	// Config Values 
	mcHomingMode 		: MC_HomingMode ; 
	fHomePosition		: LREAL := 0 ; // set position at homing
	fSafeVeloLimit		: LREAL	:= 360 ; // safe velocity limit [deg/sec]
	nEncTurnoverVal 	: LREAL ; // encoder turnover value 
	tDisabledelay		: TIME 	; // Axis idle time before axis is disabled 
END_VAR
VAR 
	bActVeloReadValid 	: BOOL ; // velocity parameter read is valid 
	bActAccReadValid 	: BOOL ; // Acceleration parameter read is valid 
	bActDecReadValid 	: BOOL ; // Deceleration parameter read is valid 
	bActParamValid 		: BOOL ; // Parameter read is valid 
END_VAR
// ===== Message data set =====
	stFault.LocationName  	:= sName 	;
	stFault.LocationNumber 	:= sNumber 	;
	stFault.ComponentType		:= E_ComponentTypes.Axis ;
	
// ===== Read system configuration =====
	McReadSysVelo	(	Axis 			:= AxisRef,
						Enable 			:= Cmd_EnDriveParRead ,
						ParameterNumber := MaxVelocitySystem ,
						ReadMode		:= 1,
						Valid			=> bActVeloReadValid ,						
						Busy			=> ,
						Error			=> ,
						ErrorID			=> ,
						Value			=> fMaxVelo );
	McReadSysAcc	(	Axis 			:= AxisRef,
						Enable 			:= Cmd_EnDriveParRead ,
						ParameterNumber := MaxAccelerationSystem ,
						ReadMode		:= 1,
						Valid			=> bActAccReadValid ,						
						Busy			=> ,
						Error			=> ,
						ErrorID			=> ,
						Value			=> fMaxAcc );
	McReadSysDec	(	Axis 			:= AxisRef,
						Enable 			:= Cmd_EnDriveParRead ,
						ParameterNumber := MaxDecelerationSystem ,
						ReadMode		:= 1,
						Valid			=> bActDecReadValid ,						
						Busy			=> ,
						Error			=> ,
						ErrorID			=> ,
						Value			=> fMaxDec );

	IF 	fMaxVelo > 0 
	AND fMaxAcc >0
	AND fMaxDec >0 THEN 
		bActParamValid	:= TRUE ; 
		fCmdAcc 		:= fMaxAcc * 0.9;
		fCmdDecc		:= fMaxDec * 0.9;
	END_IF

	IF NOT Cmd_EnDriveParRead AND NOT bActParamValid THEN  
		Cmd_EnDriveParRead := TRUE;
	ELSIF Cmd_EnDriveParRead THEN
		Cmd_EnDriveParRead := FALSE;
	END_IF

// ===== Configure Axis =====
	// ***** Config Bits *****
		THIS^.bIcfCmdVelocityRpm	:= bIcfCmdVelocityRpm	; // Enable speed inputs in Rpm
		THIS^.bIcfEnableForward 	:= bIcfEnableForward 	; // Enable forward motion
		THIS^.bIcfEnablereverse		:= bIcfEnablereverse	; // Enable reverse motion
		THIS^.bIcfAlwaysEnable		:= bIcfAlwaysEnable		; // Always enable motor and brake if safety is ok
	// ***** config homing Mode ***** 
 		THIS^.mcHomingMode 			:= mcHomingMode ; // set homing mode
		THIS^.fHomePosition			:= fHomePosition;
	// ***** Velocity settings *****
		THIS^.fSafeVeloLimit 		:= fSafeVeloLimit ; // set maximum safe velocity	
	// ***** Encoder values *****
		THIS^.fEncoderTurnoverValue := nEncTurnoverVal	; // turnover value for encoder = 25.6 mm per rev * 4096 revolutions 
	// ***** Time delay enable off *****
		THIS^.tDisableDelay 	:= tDisabledelay ;		

// ===== reset axis state indicators ======
	bError 	:= FALSE;

// ====== Set init to done =======
IF bActParamValid THEN 
	bInitDone	:= TRUE ; 
END_IF
END_METHOD

METHOD PRIVATE ExecGearDynamic : BOOL
VAR_INPUT
END_VAR
// ===== invert gear ratio if reverse slave is active =====
	IF bReverseSlave THEN 
		fbMcGearInDyn.GearRatio := fCmdGearRatio * -1 ;
	ELSE 
		fbMcGearInDyn.GearRatio := fCmdGearRatio ;
	END_IF

// ===== Execute gear in function =====
	fbMcGearInDyn ( 	Master 			:= refMasterAxis,
						Slave			:= AxisRef,
						Enable 			:= bExec_GearSlaveDyn,
						Acceleration	:= fCmdAcc	); 
						
// ===== reset command =====
	bGearedAsSlave		:= fbMcGearInDyn.InGear ; 

// Gearing fault handling 
	IF fbMcGearInDyn.Error THEN 
		bError					:= TRUE							;
		stFault.Active 			:= TRUE 						;
		stFault.MessageNumber	:= E_MessageNumbers.FF_AxisFault;
		stFault.Discription		:= CONCAT('Gear dynamic Fault ', UDINT_TO_STRING(fbMcGearInDyn.ErrorID));				;
		stFault.FaultType		:= E_FaultTypes.FF				;
		refFbFault.CmdAddFault( stFault );
	END_IF
END_METHOD

METHOD PRIVATE ExecGearIn : BOOL
VAR_INPUT
END_VAR
// ===== invert gear ratio if reverse slave is active =====
	IF bReverseSlave THEN 
		fbMcGearInSlave.RatioNumerator := fCmdGearRatio * -1 ;
	ELSE 
		fbMcGearInSlave.RatioNumerator := fCmdGearRatio ;
	END_IF

// ===== Execute gear in function =====
	fbMcGearInSlave ( 	Master 			:= refMasterAxis,
						Slave			:= AxisRef,
						Execute 		:= bExec_GearAsSlave,
						RatioDenominator:= 1	); 
						
// ===== reset command =====
	bExec_GearAsSlave 	:= FALSE  ;
	bGearedAsSlave		S= fbMcGearInSlave.InGear ; 

// Gearing fault handling 
	IF fbMcGearInSlave.Error THEN 
		bError					:= TRUE							;
		stFault.Active 			:= TRUE 						;
		stFault.MessageNumber	:= E_MessageNumbers.FF_AxisFault;
		stFault.Discription		:= CONCAT('Gear as slave Fault ', UDINT_TO_STRING(fbMcGearInSlave.ErrorID));				;
		stFault.FaultType		:= E_FaultTypes.FF				;
		refFbFault.CmdAddFault( stFault );
	END_IF
END_METHOD

METHOD PRIVATE ExecGearOut : BOOL
VAR_INPUT
END_VAR
// ===== execute gear out function ======
	fbMcGearOutSlave (	Slave 	:= AxisRef,
						Execute := bExec_GearOutSlave );

// ===== reset command =====
	bExec_GearOutSlave	:= false ;
	bGearedAsSlave		R= fbMcGearOutSlave.Done 	; 

// Gearing fault handling 
	IF fbMcGearOutSlave.Error THEN 
		bError					:= TRUE							;
		stFault.Active 			:= TRUE 						;
		stFault.MessageNumber	:= E_MessageNumbers.FF_AxisFault;
		stFault.Discription		:= CONCAT('Gear out Fault ', UDINT_TO_STRING(fbMcGearOutSlave.ErrorID));				;
		stFault.FaultType		:= E_FaultTypes.FF				;
		refFbFault.CmdAddFault( stFault );
	END_IF
END_METHOD

METHOD PRIVATE ExecHalt : BOOL
VAR_INPUT
END_VAR
// ==== Execute halt function ===== 
fbMcHalt (	Axis 		:= AxisRef,
			Execute 	:= bExec_Halt );

// ===== reset command =====
	bExec_Halt := FALSE ;
	
// Halt fault handling 
	IF fbMcHalt.Error THEN 
		bError					:= TRUE							;
		stFault.Active 			:= TRUE 						;
		stFault.MessageNumber	:= E_MessageNumbers.FF_AxisFault;
		stFault.Discription		:= CONCAT('Halt Fault ', UDINT_TO_STRING(fbMcHalt.ErrorID));				;
		stFault.FaultType		:= E_FaultTypes.FF				;
		refFbFault.CmdAddFault( stFault );
	END_IF
END_METHOD

METHOD PRIVATE ExecHome : BOOL
VAR_INPUT
END_VAR
// ==== execute homing function =====
	fbMcHome(	Axis			:= AxisRef,
				Execute			:= bExec_Home,
				HomingMode		:= mcHomingMode,
				bCalibrationCam	:= IAxisHome ); 
			
// Reset exec command 
	bExec_Home 	:= FALSE ;
	bHomed		S= fbMcHome.Done ;	
				
// fault handling 
	IF fbMcHome.Error THEN 
		bError					:= TRUE							;
		stFault.Active 			:= TRUE 						;
		stFault.MessageNumber	:= E_MessageNumbers.FF_AxisFault;
		stFault.Discription		:= CONCAT('Homing Fault ', UDINT_TO_STRING(fbMcHome.ErrorID));				;
		stFault.FaultType		:= E_FaultTypes.FF				;
		refFbFault.CmdAddFault( stFault );
	END_IF
END_METHOD

METHOD PRIVATE ExecJog : BOOL
VAR_INPUT
END_VAR
// ===== Execute Jog function =====
	// velocity limiting
		IF bCmdSafeSpeed THEN 
			fbMcJog.Velocity := MIN(fSafeVeloLimit, fbMcJog.Velocity); 
		ELSIF bCmdLimitVelocity THEN 
			fbMcJog.Velocity := MIN(fCmdVelocityLimit, fbMcJog.Velocity); 
		END_IF
	// function call
	fbMcJog (	Axis 		:= AxisRef,
				JogForward	:= bExec_JogPositive,
				JogBackwards:= bExec_JogNegative,
				Acceleration:= fCmdAcc,
				Deceleration:= fCmdDecc );

// ===== reset command =====
	bExec_JogPositive 	:= FALSE  ;
	bExec_JogNegative	:= FALSE  ;
	
// Jog fault handling 
	IF fbMcJog.Error THEN 
		bError					:= TRUE							;
		stFault.Active 			:= TRUE 						;
		stFault.MessageNumber	:= E_MessageNumbers.FF_AxisFault;
		stFault.Discription		:= CONCAT('Jog Fault ', UDINT_TO_STRING(fbMcJog.ErrorID));				;
		stFault.FaultType		:= E_FaultTypes.FF				;
		refFbFault.CmdAddFault( stFault );
	END_IF
END_METHOD

METHOD PRIVATE ExecMoveAbsolute : BOOL
VAR_INPUT
END_VAR
// ==== execute move absolute function =====
FOR i := 0 TO 1 DO 
	// velocity limiting
		IF bCmdSafeSpeed THEN 
			fbMcMoveAbsolute[i].Velocity := MIN(fSafeVeloLimit, fbMcMoveAbsolute[i].Velocity); 
		ELSIF bCmdLimitVelocity THEN 
			fbMcMoveAbsolute[i].Velocity := MIN(fCmdVelocityLimit, fbMcMoveAbsolute[i].Velocity); 
		END_IF
	// function call
	fbMcMoveAbsolute[i](	Axis 		:= AxisRef,
							Execute 	:= arExec_MoveAbs[i],
							Acceleration:= fCmdAcc,
							Deceleration:= fCmdDecc );  
	// reset Exec command 
	arExec_MoveAbs[i] := FALSE ; 

	// If function is done then reset command values
	IF fbMcMoveAbsolute[i].Done THEN 
		fbMcMoveAbsolute[i].Velocity	:= 0 ;
		fbMcMoveAbsolute[i].Position	:= 0 ; 
	END_IF
	
	// fault handling 
	IF fbMcMoveAbsolute[i].Error THEN 
		bError					:= TRUE							;
		stFault.Active 			:= TRUE 						;
		stFault.MessageNumber	:= E_MessageNumbers.FF_AxisFault;
		stFault.Discription		:= CONCAT('Move absolute Fault ', UDINT_TO_STRING(fbMcMoveAbsolute[i].ErrorID));				;
		stFault.FaultType		:= E_FaultTypes.FF				;
		refFbFault.CmdAddFault( stFault );
	END_IF
END_FOR
END_METHOD

METHOD PRIVATE ExecMoveModulo : BOOL
VAR_INPUT
END_VAR
// ===== Execute move modulo function =====
FOR i := 0 TO 1 DO 
	// velocity limiting
		IF bCmdSafeSpeed THEN 
			fbMcMoveModulo[i].Velocity := MIN(fSafeVeloLimit, fbMcMoveModulo[i].Velocity); 
		ELSIF bCmdLimitVelocity THEN 
			fbMcMoveModulo[i].Velocity := MIN(fCmdVelocityLimit, fbMcMoveModulo[i].Velocity); 
		END_IF
	// function call
	fbMcMoveModulo[i](	Axis 		:= AxisRef,
						Execute 	:= arExec_MoveModulo[i],
						Acceleration:= fCmdAcc,
						Deceleration:= fCmdDecc);  
	// reset Exec command 
	arExec_MoveModulo[i] := FALSE ; 
	
	// If function is done then reset command values
	IF fbMcMoveModulo[i].Done THEN 
		fbMcMoveModulo[i].Velocity	:= 0 ;
		fbMcMoveModulo[i].Position	:= 0 ; 
	END_IF
	
	// fault handling 
	IF fbMcMoveModulo[i].Error THEN 
		bError					:= TRUE							;
		stFault.Active 			:= TRUE 						;
		stFault.MessageNumber	:= E_MessageNumbers.FF_AxisFault;
		stFault.Discription		:= CONCAT('Move module Fault ', UDINT_TO_STRING(fbMcMoveModulo[i].ErrorID));				;
		stFault.FaultType		:= E_FaultTypes.FF			;
		refFbFault.CmdAddFault( stFault );
	END_IF
END_FOR
END_METHOD

METHOD PRIVATE ExecMoveRelative : BOOL
VAR_INPUT
END_VAR
// ===== Execute move relative function ======
FOR i := 0 TO 1 DO 
	// velocity limiting
		IF bCmdSafeSpeed THEN 
			fbMCMoveRelative[i].Velocity := MIN(fSafeVeloLimit, fbMCMoveRelative[i].Velocity); 
		ELSIF bCmdLimitVelocity THEN 
			fbMCMoveRelative[i].Velocity := MIN(fCmdVelocityLimit, fbMCMoveRelative[i].Velocity); 
		END_IF
	// function call
	fbMCMoveRelative[i](	Axis 		:= AxisRef,
							Execute		:= arExec_MoveRelative[i],
							Acceleration:= fCmdAcc,
							Deceleration:= fCmdDecc );
	// reset Exec command 
	arExec_MoveRelative[i] := FALSE ; 

	// If function is done then reset command values
	IF fbMCMoveRelative[i].Done THEN 
		fbMCMoveRelative[i].Velocity	:= 0 ;
		fbMCMoveRelative[i].Distance	:= 0 ; 
	END_IF
	
	// fault handling 
	IF fbMCMoveRelative[i].Error THEN 
		bError					:= TRUE							;
		stFault.Active 			:= TRUE 						;
		stFault.MessageNumber	:= E_MessageNumbers.FF_AxisFault;
		stFault.Discription		:= CONCAT('Move relative Fault ', UDINT_TO_STRING(fbMCMoveRelative[i].ErrorID));				;
		stFault.FaultType		:= E_FaultTypes.FF			;
		refFbFault.CmdAddFault( stFault );
	END_IF
END_FOR
END_METHOD

METHOD PRIVATE ExecMoveVelocity : BOOL
VAR_INPUT
END_VAR
// ===== Execute move velocity function =====
// velocity limiting
IF bCmdSafeSpeed THEN 
	fbMcMoveVelocity.Velocity := MIN(fSafeVeloLimit, fbMcMoveVelocity.Velocity); 
ELSIF bCmdLimitVelocity THEN 
	fbMcMoveVelocity.Velocity := MIN(fCmdVelocityLimit, fbMcMoveVelocity.Velocity); 
END_IF
// function call
fbMcMoveVelocity (	Axis 		:= AxisRef,
					Execute		:= bExec_MoveVelocity,
					Acceleration:= fCmdAcc,
					Deceleration:= fCmdDecc );

// ===== reset command =====
bExec_MoveVelocity := FALSE ;
	
// Halt fault handling 
IF fbMcHalt.Error THEN 
	bError					:= TRUE							;
	stFault.Active 			:= TRUE 						;
	stFault.MessageNumber	:= E_MessageNumbers.FF_AxisFault;
	stFault.Discription		:= CONCAT('Move velocity Fault ', UDINT_TO_STRING(fbMcMoveVelocity.ErrorID));				;
	stFault.FaultType		:= E_FaultTypes.FF				;
	refFbFault.CmdAddFault( stFault );
END_IF
END_METHOD

METHOD PRIVATE ExecEnable : BOOL
VAR_INPUT
END_VAR
// ===== Set axis enable ======
IF NOT bEnable AND NOT AxisRef.Status.MotionCommandsLocked THEN
	bCmdSafeStop	S= TRUE ;
ELSE 
	bCmdEnableAxis	:= bEnable ;
END_IF

// ===== Check if axis is bussy with a command =====
	bInternalEnable S= AxisRef.Status.HasJob;
	bInternalEnable	S= bIcfAlwaysEnable ; // always enable axis if configured
	bInternalEnable	S= AxisRef.Status.Coupled ;
	
// ===== Axis disable timer after last command =====
	TofIntAxisEnable (	IN:= bInternalEnable, PT := tDisableDelay);

// ===== Enable drive =====
	fbMcPower(	Axis			:= AxisRef , 
				Enable			:= bCmdEnableAxis AND TofIntAxisEnable.Q, 
				Enable_Positive	:= bIcfEnableForward, 
				Enable_Negative	:= bIcfEnablereverse, 
				Override		:= 100 );  
				
// ===== Reset internal enable signal =====
	bInternalEnable := FALSE ; 	

IF fbMcPower.Error THEN 
	bError					:= TRUE							;
	stFault.Active 			:= TRUE 						;
	stFault.MessageNumber	:= E_MessageNumbers.FF_AxisFault;
	stFault.Discription		:= CONCAT('Enable Fault ', UDINT_TO_STRING(fbMcPower.ErrorID));				;
	stFault.FaultType		:= E_FaultTypes.FF				;
	refFbFault.CmdAddFault( stFault );
END_IF
END_METHOD

METHOD PRIVATE ExecReadStatus : BOOL
VAR_INPUT
END_VAR
// Read axis status from drive
fbMcReadAxisStatus (	Enable 	:= TRUE ,
						Axis 	:= AxisRef );
						
// convert velocity to RPM for output if aplicable
IF bIcfCmdVelocityRpm THEN 
	fVelocity := AxisRef.NcToPlc.ActVelo / 6 ;
ELSE 
	fVelocity := AxisRef.NcToPlc.ActVelo ;
END_IF
						
// set status bits 
bIdle := NOT AxisRef.Status.HasJob ;

// read fault handling 
IF fbMcReadAxisStatus.Error THEN 
	bError					:= TRUE							;
	stFault.Active 			:= TRUE 						;
	stFault.MessageNumber	:= E_MessageNumbers.FF_AxisFault;
	stFault.Discription		:= CONCAT('Status read fault ', UDINT_TO_STRING(fbMcPower.ErrorID));				;
	stFault.FaultType		:= E_FaultTypes.FF				;
	refFbFault.CmdAddFault( stFault );
END_IF
END_METHOD

METHOD PRIVATE ExecReset : BOOL
VAR_INPUT
END_VAR
IF  AxisRef.Status.Moving THEN // If the axis is still moving execute safe stop first
	CmdSafeStop();
	RETURN;
END_IF

// ===== Reset axis, drive and axis functions =====
	fbSoeReset ( 	Execute := bExec_Reset AND NOT fbMcReset.Busy AND NOT bIcfSimulationMode, // No physical drive reset necesarry when not connected 
					Timeout := T#10S		,
					Axis	:= AxisRef		);
	
	fbMcReset	( 	Execute	:= bexec_reset AND NOT fbSoeReset.Busy,
					Axis	:= AxisRef ); 
					
// ===== reset command =====
	bExec_Reset := FALSE ;
	
// ===== reset internal fault bits and stop bits =====
	bError 			:= FALSE ; 
	
// ===== reset safe commands ======
	bCmdSafeStop	:= FALSE ; 
	bCmdSafeSpeed 	:= FALSE ;
	
// Reset fault handling 
	IF fbSoeReset.Error OR fbMcReset.Error THEN 
		bError					:= TRUE							;
		stFault.Active 			:= TRUE 						;
		stFault.MessageNumber	:= E_MessageNumbers.FF_AxisFault;
		stFault.Discription		:= CONCAT('Reset Fault ', UDINT_TO_STRING(fbMcReset.ErrorID))			;
		stFault.FaultType		:= E_FaultTypes.FF				;
		refFbFault.CmdAddFault( stFault );
	END_IF
END_METHOD

METHOD PRIVATE ExecSafeFunctions : BOOL
VAR_INPUT
END_VAR
// ==== Safe operation functions (overrule all other motion functions) =====
	fbMcStop( 	Axis 			:= AxisRef		,
				Execute 		:= bCmdSafeStop	,
				Deceleration	:= fMaxDec		);
	
	// Reset axis command			
	bCmdSafeStop 	R= fbMcStop.Done OR AxisRef.Status.HasBeenStopped ;
	bStopped		:= AxisRef.Status.HasBeenStopped ;
	
// Safestop fault handling 
	IF fbMcStop.Error THEN 
		bError					:= TRUE							;
		stFault.Active 			:= TRUE 						;
		stFault.MessageNumber	:= E_MessageNumbers.FF_AxisFault;
		stFault.Discription		:= CONCAT('Safe stop axis fault ', UDINT_TO_STRING(fbMcStop.ErrorID));				;
		stFault.FaultType		:= E_FaultTypes.FF				;
		refFbFault.CmdAddFault( stFault );
	END_IF
	
// ===== Safe speed monitoring =====
	IF bCmdSafeSpeed THEN 
		IF AxisRef.NcToPlc.ActVelo > fSafeVeloLimit THEN 
			bExec_Halt := TRUE ; 
			ExecHalt(); 
		ELSE 
			bCmdSafeSpeed := FALSE ; 
		END_IF
	END_IF

// ===== Dev is safe feedback =====
bDevIsSafe := AxisRef.Status.HasBeenStopped AND NOT bCmdEnableAxis ;
END_METHOD

METHOD PRIVATE METH_ExecuteMotionFunctions : BOOL
VAR_INPUT
END_VAR
// ===== Check if safe to move =====
	IF bCmdSafeStop THEN 
		RETURN ;
	END_IF

// ===== Homing functions =====
	ExecHome		(); 

// ===== Motion standstil commands =====
	ExecHalt		();

// ===== Motion move functions
	ExecJog			(); 
	ExecMoveAbsolute();
	ExecMoveRelative();
	ExecMoveModulo	();
	ExecMoveVelocity();
	
// ===== Execute gearing functions =====
	ExecGearIn		();
	ExecGearDynamic	();
	ExecGearOut		();
	
// ====== reset velocity lmiting =====
	bVelocityLimited	:= bCmdLimitVelocity ;	
	bCmdLimitVelocity 	:= FALSE ;
END_METHOD

METHOD PRIVATE METH_ExecuteOrganizationFunctions : BOOL
VAR_INPUT
END_VAR
// ==== execute organizational functions =====
	ExecReadStatus	(); 
	ExecEnable		();
	ExecReset		();
END_METHOD

END_FUNCTION_BLOCK

// Buttons/Functions/FB_DevHMIButton
FUNCTION_BLOCK PUBLIC FB_DevHMIButton EXTENDS FB_DevBase // Button function for HMI 
VAR_INPUT
	Istatus			: BOOL	:= FALSE;// Digital sensor, Direct input status
	tDelay			: TIME 	:= T#5S	;// Time before delayed signal becomes active 
	bCmdSimulate	: BOOL 	:= FALSE;// Simulate sensor Input 
	bSimState		: BOOL 	:= FALSE;// Simulated sensor state
END_VAR
VAR_OUTPUT
	bFcoInputActive		: BOOL 			;// Digital sensor, Button active state
	bFcoDelay			: BOOL			;// Button, Delayed input status (3 seconds) 
	bFeStatus			: BOOL			;// Button, Falling edge of input signal	
	bReStatus			: BOOL			;// Button, Rising edge of input signal
	TetInputActive		: TIME			;// Button, Time elapsed while button is active
	bInvisible			: BOOL 			;// Button, Button is made invisible
	bDeactivate			: BOOL 			;// Button, Deactivate button 
END_VAR
VAR
	FB_delIStatus: TON; // Timer function for delayed input status 
	FB_feIStatus: F_TRIG; // generate falling edge pulse edge from Istatus
	FB_reIStatus: R_TRIG; // generate falling edge pulse edge from Istatus
END_VAR

// ***** Direct input when enabled *****
IF bEnable THEN 
	IF bCmdSimulate  THEN 
		bFcoInputActive := bSimState ; 
	ELSE
		bFcoInputActive := Istatus ;
	END_IF
ELSE 
	bFcoInputActive := FALSE ;
END_IF

// ===== check if function is enabled =====
	IF NOT bEnable THEN 
		bInvisible 	:= TRUE ;
		bDeactivate	:= TRUE ;
		bFcoDelay	:= FALSE;
		RETURN;
	ELSE  
		bInvisible 	:= FALSE ;
		bDeactivate	:= FALSE ;
	END_IF

// ====== process functions if enabled ======
	// ***** Set Delayed inputs and time elapsed ****
		FB_delIStatus(	IN:= bFcoInputActive,
						PT:= tDelay , 
						Q=> bFcoDelay , 
						ET=> TetInputActive 
					  ); // Generate delayed input status from push button input status
	// ***** Edge triggers *****
		FB_feIStatus(CLK:= Istatus , Q=> bFeStatus ); // generate falling edge pulse on pushbutton input
		FB_reIStatus (Clk := Istatus , Q => bReStatus); // Generate rising edge from push button input signal

END_FUNCTION_BLOCK

// Buttons/Functions/FB_DevPushButton
FUNCTION_BLOCK PUBLIC FB_DevPushButton EXTENDS Fb_DevDigitalInputFunctions
VAR_INPUT
END_VAR
VAR_OUTPUT
END_VAR
VAR
END_VAR

SUPER^();

END_FUNCTION_BLOCK

// Buttons/Functions/FB_DevPushbuttonLight
FUNCTION_BLOCK PUBLIC FB_DevPushbuttonLight EXTENDS FB_DevPushButton
VAR_INPUT
	sCmdLightState	: E_LightState ; // feedback lights status 
END_VAR
VAR_OUTPUT
END_VAR
VAR
	fbLight : Fb_DevLight ; // light control 
END_VAR

SUPER^();

// Light commands
	CASE sCmdLightState OF
		Light_Off:
			fbLight.eCmdLight := E_LightState.Light_Off;
		Light_BlinkSlow:
			fbLight.eCmdLight := E_LightState.Light_BlinkSlow ;
		Light_BlinkFast:
			fbLight.eCmdLight := E_LightState.Light_BlinkFast ;
		Light_On:
			fbLight.eCmdLight := E_LightState.Light_On ;
	END_CASE
	
fbLight(bEnable := TRUE);

END_FUNCTION_BLOCK

// Lights/Functions/Fb_DevLight
FUNCTION_BLOCK PUBLIC Fb_DevLight
VAR_INPUT
	bEnable			: BOOL	:= TRUE ;// Enable light
	eCmdLight		: E_LightState := E_LightState.Light_Off ; // commanded light state [Light_off, _On, _BlinkFast, _BlinkSlow]
END_VAR
VAR_OUTPUT
END_VAR
VAR
	qLight AT %Q* : BOOL := FALSE ; // light output
END_VAR

// ===== check if light is enabled ======
	IF NOT bEnable THEN 
		qLight := FALSE ;
		RETURN; 
	END_IF
	
// ===== set light output ======
	Mod_SetOutput();

METHOD PRIVATE Mod_SetOutput : BOOL
VAR_INPUT
END_VAR
// ===== set light output state =====
	CASE eCmdLight OF
		Light_BlinkSlow:
			qLight := Sys_Variables.BlinkSlow ;
		Light_BlinkFast:
			qLight	:= Sys_Variables.BlinkFast ;
		Light_On:
			qLight := TRUE ;
		ELSE
			qLight := FALSE ;
	END_CASE
END_METHOD

END_FUNCTION_BLOCK

// Encoders/FunctionBlocks/FB_EncoderBase
FUNCTION_BLOCK PUBLIC FB_EncoderBase
VAR_INPUT
	nCfgUnitsPerPulse	: LREAL := 1	; // Scale factor for output [units/pulse]
	nCfgOffset			: LREAL := 0	; // Offset for output
	
	bIcfInverted		: BOOL	:= FALSE; // Invert output position = standard false  
END_VAR
VAR_OUTPUT
	nOutPosition		: LREAL	:= 0	; // Scaled position output
	nOutRaw				: UDINT := 0	; // Raw output value	 
	nVelocity			: LREAL	:= 0 	; // Velocity [units/sec]
END_VAR
VAR
END_VAR

METHOD PUBLIC FastTask : BOOL
VAR_INPUT
END_VAR
END_METHOD

END_FUNCTION_BLOCK

// Encoders/FunctionBlocks/FB_EncoderInput
FUNCTION_BLOCK FB_EncoderInput EXTENDS FB_EncoderBase
VAR_INPUT
END_VAR
VAR_OUTPUT
END_VAR
VAR
	iEncoderSignal AT%I*: UDINT ;
	
	nScaledValue		: LREAL ; // Only scaled value for internal use
	nValueWithOffset	: LREAL ; // scaled value with added offset
END_VAR

// ====== Scale Output value ======
	nScaledValue := UDINT_TO_LREAL(iEncoderSignal) * nCfgUnitsPerPulse ;

// ====== Invert ======
	IF bIcfInverted THEN 
		nScaledValue := nScaledValue * -1;
	END_IF
	
// ====== Add offset ======= 
	nValueWithOffset := nScaledValue + nCfgOffset ;

// ====== Set Outputs =======
	nOutPosition 	:= nValueWithOffset ;
	nOutRaw			:= iEncoderSignal	;

METHOD PUBLIC FastTask : BOOL
VAR_INPUT
END_VAR
END_METHOD

END_FUNCTION_BLOCK

// GroupHandlers/ManualControlHandler/FB_DevManualHandler
FUNCTION_BLOCK FB_DevManualHandler
VAR_INPUT
END_VAR
VAR_OUTPUT
END_VAR
VAR
END_VAR

END_FUNCTION_BLOCK

// Heaters/FB_DevPWMGenerator
FUNCTION_BLOCK PUBLIC FB_DevPWMGenerator EXTENDS FB_DevBase
VAR_INPUT
	nPeriodLength		: DINT	:= 2000 	; // desired PWM cycle time length [ms] 
	nDutyCycle 	: DINT	:= 0 		; // percentage of power 
END_VAR
VAR_OUTPUT
END_VAR
VAR
	qbOutput	AT %Q* 	: BOOL 	; // physical output
	bCycleOutput		: BOOL 	; // Cycle output
	tonTimerOn  		: TON 	; // Timer for cycle on
	tofTimerOff			: TOF 	; // timer for cycle off 
	// output commands
	bCmdPWMCycle		: BOOL 	; // run PWM cycle 
	bCmdOn				: BOOL 	; // turn output on permanantly
	
END_VAR

// check for enable
IF NOT bEnable THEN 
	qbOutput := FALSE ;
	RETURN; 
ELSE 
	SUPER^(); 
END_IF

// calculate cycle times 
CalcCycle();
// set outputs
ExecSetOutput();

METHOD PRIVATE CalcCycle : BOOL
VAR_INPUT
END_VAR
// check if dutycycle is within limits
nDutyCycle := LIMIT(1,nDutyCycle,100);

// Calculate time on from cycle time
tonTimerOn.PT 	:= DINT_TO_TIME(( nPeriodLength / 100) * nDutyCycle);
tofTimerOff.PT	:= DINT_TO_TIME(( nPeriodLength / 100) * (100 - nDutyCycle));
END_METHOD

METHOD PRIVATE ExecSetOutput : BOOL
VAR_INPUT
END_VAR
// PWM signal generator
IF bCmdPWMCycle THEN 
	// Run cycle timers 
	tofTimerOff	(IN := tonTimerOn.Q);
	tonTimerOn	(IN := bCycleOutput AND NOT tofTimerOff.Q );
	bCycleOutput := NOT tofTimerOff.Q ;
ELSE
	bCycleOutput := FALSE ;
END_IF

// set output 
qbOutput := bCycleOutput OR bCmdOn ;

// reset continuous on command
bCmdOn := false ;
END_METHOD

METHOD PUBLIC CmdOutputCycle : BOOL // start PWM cycle stays on until off command is given
VAR_INPUT
END_VAR
bCmdPWMCycle 	S= TRUE ;
CmdOutputCycle 	:= bCmdPWMCycle ;
END_METHOD

METHOD PUBLIC CmdOutputOff : BOOL // turn off output signal completely
VAR_INPUT
END_VAR
bCmdPWMCycle 	:= FALSE ;
bCmdOn			:= FALSE ;
CmdOutputOff	:= TRUE 	;
END_METHOD

METHOD PUBLIC CmdOutputOn : BOOL // Output stays on until command ends (returns to PWM if active otherwise turns off)
VAR_INPUT
END_VAR
bCmdOn 		S= TRUE ;
CmdOutputOn	:= TRUE ;
END_METHOD

END_FUNCTION_BLOCK

// Outputs/DigitalOutputs/FB_DigitalOutput
FUNCTION_BLOCK PUBLIC FB_DigitalOutput EXTENDS FB_DevBase
VAR_INPUT
	bCmdOn	: BOOL := FALSE ; // command output status
END_VAR
VAR_OUTPUT
	bOutputState	: BOOL := FALSE ; // State of physical output
END_VAR
VAR
	qbOutput AT%Q* : BOOL ; // Output to physical device
END_VAR

METHOD PRIVATE ExecSetFeedback : BOOL
VAR_INPUT
END_VAR
// Set feedback 
bOutputState := qbOutput ;
END_METHOD

METHOD PRIVATE ExecSetOutput : BOOL
VAR_INPUT
END_VAR
// Set Output to physical device
IF bEnable THEN 
	qbOutput := bCmdOn ; 
ELSE 
	qbOutput S= FALSE ; 
END_IF

bCmdOn := false ;
END_METHOD

METHOD PUBLIC CmdOn : BOOL
VAR_INPUT
END_VAR
bCmdOn S= TRUE ; 

CmdOn := bOutputState ;
END_METHOD

END_FUNCTION_BLOCK

// Sensors/FootPedals/FunctionBlocks/FB_EfkaEB301A_FootPedal
FUNCTION_BLOCK PUBLIC FB_EfkaEB301A_FootPedal
VAR_INPUT
	bEnable : BOOL := TRUE ;
END_VAR
VAR_OUTPUT
	ePedalInputStep		: E_FootpedalPos	:= 0 ;
	bRTrigtoReverse1 	: BOOL := FALSE ; // rising edge trigger when pedal moves from 0 to -1 or Idle to reverse 1 
	bRTrigtoReverse2 	: BOOL := FALSE ; // rising edge trigger when pedal moves from 1 to -2 or reverse 1 to reverse 2 
	bRTrigtoForward1 	: BOOL := FALSE ; // rising edge trigger when pedal moves from 0 to 1 or idle to forward 1 
	bRTrigtoForward2 	: BOOL := FALSE ; // rising edge trigger when pedal moves from 0 to 1 or forward to forward 2 
END_VAR
VAR
	// ===== greycode switches from footpedal =====
	I_GreyCodeA AT%I* : BOOL	; // Greycode input a from foot pedal 
	I_GreyCodeB AT%I* : BOOL	; // Greycode input a from foot pedal 
	I_GreyCodeC AT%I* : BOOL	; // Greycode input a from foot pedal 
	I_GreyCodeD AT%I* : BOOL	; // Greycode input a from foot pedal 
	nGreyCodetotal	: BYTE ; // all greycode switches combined
	// ==== decimal value =====
	ePreviousPedalInput	: E_FootpedalPos	:= 0 ;
END_VAR

// ===== Read input from pedal =====
ACT_ConvertGreycode();

// ===== Create edge flanks for functions =====
ACT_CreateEdges();

ACTION ACT_ConvertGreycode:
// ===== Combine greycode sensors =====
nGreyCodetotal.0 := I_GreyCodeA ;
nGreyCodetotal.1 := I_GreyCodeB ;
nGreyCodetotal.2 := I_GreyCodeB ;
nGreyCodetotal.3 := I_GreyCodeC ;

// ==== Convert greycode decimal to speed steps =====
// this only makes sense in EFKA world but anyway let's convert it to our own sense
CASE nGreyCodetotal OF 
	12: ePedalInputStep := E_FootpedalPos.eReverse1	;
	14: ePedalInputStep := E_FootpedalPos.eReverse2	;
	15: ePedalInputStep := E_FootpedalPos.eIdle		;
	13: ePedalInputStep := E_FootpedalPos.eForward1	;
	09: ePedalInputStep := E_FootpedalPos.eForward2	;
 	08: ePedalInputStep := E_FootpedalPos.eForward3	;
	10: ePedalInputStep := E_FootpedalPos.eForward4	;
	11: ePedalInputStep := E_FootpedalPos.eForward5	;
	03:	ePedalInputStep := E_FootpedalPos.eForward6	;
	02:	ePedalInputStep := E_FootpedalPos.eForward7	;
	00: ePedalInputStep := E_FootpedalPos.eForward8	;
	01: ePedalInputStep := E_FootpedalPos.eForward9	;
	05: ePedalInputStep := E_FootpedalPos.eForward10	;
	04: ePedalInputStep := E_FootpedalPos.eForward11	;
	06: ePedalInputStep := E_FootpedalPos.eForward12 	;
	07: ePedalInputStep := E_FootpedalPos.eForward13	;
	ELSE
		ePedalInputStep := E_FootpedalPos.eFalse 		;
END_CASE
END_ACTION

ACTION ACT_CreateEdges:
// ===== create edges on which functions can be triggerd =====
CASE ePedalInputStep OF
	E_FootpedalPos.eReverse2:
		bRTrigtoReverse2 := ePreviousPedalInput = E_FootpedalPos.eReverse1 ;
	E_FootpedalPos.eReverse1:
		bRTrigtoReverse1 := ePreviousPedalInput = E_FootpedalPos.eIdle ;
	E_FootpedalPos.eForward1:
		bRTrigtoForward1 := ePreviousPedalInput = E_FootpedalPos.eIdle ;
	E_FootpedalPos.eForward2: 
		bRTrigtoForward2 := ePreviousPedalInput = E_FootpedalPos.eForward1 ; 
END_CASE 

// write previous pedal input 
ePreviousPedalInput := ePedalInputStep ;
END_ACTION

END_FUNCTION_BLOCK
